PROGRAM MAIN
VAR
END_VAR

PRG_DecoSample();
PRG_MOVE();

END_PROGRAM

(* stored: Version 1.1.0.1, ProductVersion 3.1.4026.6
   POU MAIN: Id {66350254-5d0d-4517-a4ad-317237f50595}, SpecialFunc None *)
